PROGRAM TESTPRG
VAR
    plcopenCommandTest : PLCopenCommand_Test;
    plcopenCallTest : PLCopenCall_Test;
END_VAR

// Copyright (c) 2024 Loupe (https://loupe.team), provided under the MIT License.

TcUnit.RUN();

END_PROGRAM

(* stored: Version 1.1.0.1
   POU TESTPRG: Id {da7b43c9-38b1-4c6f-a60e-db64ccc086f5}, SpecialFunc None *)
